// Mitsubishi GX Works2 project: LRI_PLC_27.09   PLC: Q03UDV
// PLC1_Rebcca

PROGRAM MAIN
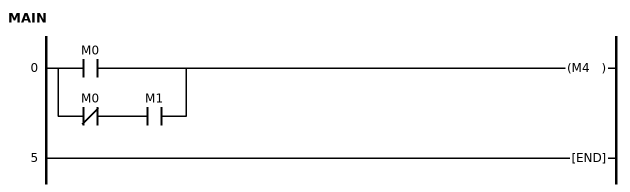
0     LD      M0
      LDI     M0
      AND     M1
      ORB
      OUT     M4
5     END
END_PROGRAM
